{attribute 'linkalways'} 
{attribute 'no_explicit_call' := 'This FB is a CLASS and must be accessed using methods or properties'}
{attribute 'enable_dynamic_creation'}
FUNCTION_BLOCK _TcVnArray8_LREAL EXTENDS AliasDatatypeBase
VAR
	localData : TcVnArray8_LREAL;
	activeData : REFERENCE TO TcVnArray8_LREAL REF= localData;
	aliasBaseDatatype : _Array0to7OfLREAL;
END_VAR

PROPERTY PUBLIC Address : PVOID
GET
Address := ADR(activeData);
END_GET
END_PROPERTY

METHOD PUBLIC ClearReference
VAR_INPUT
END_VAR
activeData REF= localData;
SetBaseDatatypeReference();
END_METHOD

METHOD PUBLIC Clone : I_Datatype
VAR
    pClone : POINTER TO _TcVnArray8_LREAL;
END_VAR
pClone := __NEW(_TcVnArray8_LREAL);
Clone := pClone^;
END_METHOD

METHOD FB_init : BOOL
VAR_INPUT
	bInitRetains : BOOL; // if TRUE, the retain variables are initialized (warm start / cold start)
	bInCopyCode : BOOL;  // if TRUE, the instance afterwards gets moved into the copy code (online change)
	//InitialValue : TcVnArray8_LREAL; // if possible, not all values can be initialized
END_VAR
//localData := InitialValue; // if possible, not all values can be initialized
SetBaseDatatypeReference();
AddBaseDatatype(aliasBaseDatatype);
END_METHOD

PROPERTY PUBLIC Identifier : T_MAXSTRING
GET
Identifier := 'TcVnArray8_LREAL';
END_GET
END_PROPERTY

METHOD PUBLIC MakeReferenceTo
VAR_INPUT
	ReferenceTarget : REFERENCE TO TcVnArray8_LREAL;
END_VAR
activeData REF= ReferenceTarget;
SetBaseDatatypeReference();
END_METHOD

METHOD PROTECTED SetBaseDatatypeReference
VAR_INPUT
END_VAR
aliasBaseDatatype.MakeReferenceTo(activeData);
END_METHOD

PROPERTY PUBLIC Size : UDINT
GET
Size := SIZEOF(activeData);
END_GET
END_PROPERTY

METHOD TryMakeReferenceTo : BOOL
VAR_INPUT
	Target : I_Datatype;
END_VAR
VAR
	targetAsAlias : I_AliasDatatype;
	pTargetData : POINTER TO TcVnArray8_LREAL;
END_VAR
IF NOT Target.TryResolveAsAliasDatatype(targetAsAlias) THEN
	RETURN;
END_IF

IF targetAsAlias.Identifier <> Identifier THEN
	RETURN;
END_IF

pTargetData := Target.Address;
activeData REF= pTargetData^;
SetBaseDatatypeReference();
TryMakeReferenceTo := TRUE;
END_METHOD

PROPERTY PUBLIC Value : REFERENCE TO TcVnArray8_LREAL
GET
Value REF= activeData;
END_GET
END_PROPERTY

END_FUNCTION_BLOCK

(* stored: Version 1.1.0.1, ProductVersion 3.1.4024.13
   POU _TcVnArray8_LREAL: Id {53a9642b-fdef-0a77-2dd1-2cf1565b21d4}, SpecialFunc None
   Folder Core: Id {66d2f21b-04d4-0289-2ace-0c514297bfcd}
   Folder Protected: Id {a9a4476d-8a9b-0f29-191d-0c8d8073824c}
   Folder Customize: Id {6d311d1e-a1c9-0c81-25b5-c29456c46a8f}
   Folder Constructor: Id {0d3c736d-ba80-0d46-3740-944fa4958533}
   Property Address: Id {94febebd-bacf-0d41-23de-dc2d9c23a35d}
   Get Get: Id {21bd5850-8e0a-043e-2241-ce4420e74eaf}
   Method ClearReference: Id {7414a532-b14d-0df6-0e23-06aedf561006}
   Method Clone: Id {08f3c3af-36c5-0ff8-2c65-daadfaa5ef3d}
   Method FB_init: Id {60fc61c3-1de9-095b-365c-3190eb58c048}
   Property Identifier: Id {c43f5e2f-ff66-0550-1ebc-3c172f3f9640}
   Get Get: Id {24c457ea-8470-05f6-17ea-4d0ba6792494}
   Method MakeReferenceTo: Id {dc12af93-4e7f-0a35-2b60-67c5b5e2ab85}
   Method SetBaseDatatypeReference: Id {1496396e-7aa0-0156-0620-ab5100276299}
   Property Size: Id {b385a9ea-99f4-0ace-0289-0b31bd9d121a}
   Get Get: Id {62a74c04-8125-0905-1f20-6d89ce031499}
   Method TryMakeReferenceTo: Id {18fe6bf6-6f8a-0a38-0e39-2950417eef09}
   Property Value: Id {b090f3ef-28d2-074d-1169-f9e520878ebf}
   Get Get: Id {6a036798-42da-06ab-1380-30317271adc2} *)
